// TIA Portal project "Practica3Equipo" (V16)

(* hardware
DEVICE "S7300/ET200M station_1"  S7-300 station
   slot 0: "Rail_0"  Rail  6ES7 390-1***0-0AA0
   slot 2: "PLC_1"  CPU 314  6ES7 314-1AG13-0AB0  V2.6
      slot 0: "MPI interface_1"  X1
*)

// ===== PLC "PLC_1"  CPU 314 =====

VAR_GLOBAL   // PLC tag table "Estados"
   "E0" AT %M0.0 : Bool;
   "E1" AT %M0.1 : Bool;
   "E2" AT %M0.2 : Bool;
   "E3" AT %M0.3 : Bool;
   "E4" AT %M0.4 : Bool;
   "E5" AT %M0.5 : Bool;
   "E6" AT %M0.6 : Bool;
   "E7" AT %M0.7 : Bool;
   "E8" AT %M1.0 : Bool;
   "E9" AT %M1.1 : Bool;
   "E10" AT %M1.2 : Bool;
   "E11" AT %M1.3 : Bool;
   "E12" AT %M1.4 : Bool;
   "E13" AT %M1.5 : Bool;
   "E14" AT %M1.6 : Bool;
   "E15" AT %M1.7 : Bool;
   "E16" AT %M2.0 : Bool;
   "E17" AT %M2.1 : Bool;
   "E18" AT %M2.2 : Bool;
   "E19" AT %M2.3 : Bool;
END_VAR

VAR_GLOBAL   // PLC tag table "Inputs"
   "P3inWork" AT %I10.0 : Bool;
   "P3inHome" AT %I10.1 : Bool;
   "P3engaged" AT %I10.2 : Bool;
   "RStation1" AT %I10.3 : Bool;
   "RStation2" AT %I10.4 : Bool;
   "Lightbarrier" AT %I10.5 : Bool;
   "inPlace3" AT %I10.6 : Bool;
   "inPlace4" AT %I10.7 : Bool;
   "P1inWork" AT %I11.0 : Bool;
   "P1inHome" AT %I11.1 : Bool;
   "P2inWork" AT %I11.2 : Bool;
   "P2inHome" AT %I11.3 : Bool;
   "P1engaged" AT %I11.4 : Bool;
   "P2engaged" AT %I11.5 : Bool;
   "inPlace1" AT %I11.6 : Bool;
   "inPlace2" AT %I11.7 : Bool;
   "chainMagnet" AT %I13.6 : Bool;
END_VAR

VAR_GLOBAL   // PLC tag table "Outputs"
   "Chain" AT %Q11.0 : Bool;
   "Belt" AT %Q11.1 : Bool;
   "P1toWork" AT %Q11.2 : Bool;
   "P1toHome" AT %Q11.3 : Bool;
   "P2toWork" AT %Q11.4 : Bool;
   "P2toHome" AT %Q11.5 : Bool;
   "P3toWork" AT %Q11.6 : Bool;
   "P3toHome" AT %Q11.7 : Bool;
END_VAR

FUNCTION "Secuencial" : Void   // FC1, LAD
{ S7_Optimized_Access := 'FALSE' }
VERSION : 0.1
   VAR_TEMP   // added for the SCL form of the ladder/FBD networks
      _w1 : Bool;
   END_VAR
BEGIN

REGION Network 1
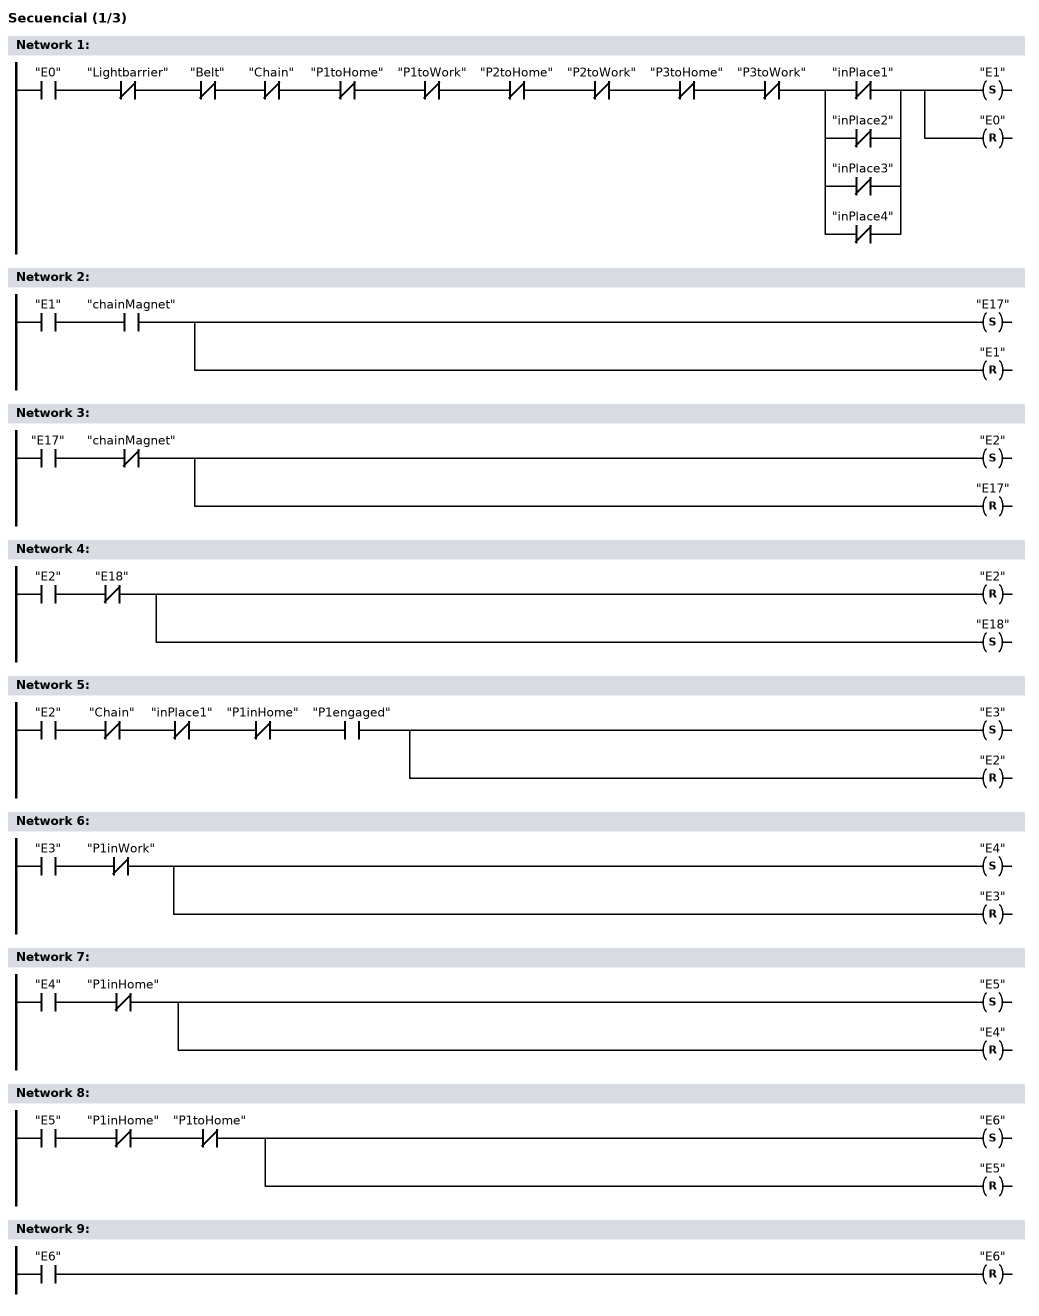
   RUNG wire#powerrail
      Contact( "E0" )
      I_Contact( "Lightbarrier" )
      I_Contact( "Belt" )
      I_Contact( "Chain" )
      I_Contact( "P1toHome" )
      I_Contact( "P1toWork" )
      I_Contact( "P2toHome" )
      I_Contact( "P2toWork" )
      I_Contact( "P3toHome" )
      I_Contact( "P3toWork" )
      wire#w1
      I_Contact( "inPlace1" )
      wire#w2
      S_Coil( "E1" )
   END_RUNG
   RUNG wire#w1
      I_Contact( "inPlace2" )
   END_RUNG wire#w2
   RUNG wire#w1
      I_Contact( "inPlace3" )
   END_RUNG wire#w2
   RUNG wire#w1
      I_Contact( "inPlace4" )
   END_RUNG wire#w2
   RUNG wire#w2
      R_Coil( "E0" )
   END_RUNG
   // the same network as SCL:
   IF "E0" AND NOT "Lightbarrier" AND NOT "Belt" AND NOT "Chain" AND NOT "P1toHome" AND NOT "P1toWork" AND NOT "P2toHome" AND NOT "P2toWork" AND NOT "P3toHome" AND NOT "P3toWork" AND (NOT "inPlace1" OR NOT "inPlace2" OR NOT "inPlace3" OR NOT "inPlace4") THEN
       "E1" := TRUE;
       "E0" := FALSE;
   END_IF;
END_REGION

REGION Network 2
   RUNG wire#powerrail
      Contact( "E1" )
      Contact( "chainMagnet" )
      wire#w1
      S_Coil( "E17" )
   END_RUNG
   RUNG wire#w1
      R_Coil( "E1" )
   END_RUNG
   // the same network as SCL:
   IF "E1" AND "chainMagnet" THEN
       "E17" := TRUE;
       "E1" := FALSE;
   END_IF;
END_REGION

REGION Network 3
   RUNG wire#powerrail
      Contact( "E17" )
      I_Contact( "chainMagnet" )
      wire#w1
      S_Coil( "E2" )
   END_RUNG
   RUNG wire#w1
      R_Coil( "E17" )
   END_RUNG
   // the same network as SCL:
   IF "E17" AND NOT "chainMagnet" THEN
       "E2" := TRUE;
       "E17" := FALSE;
   END_IF;
END_REGION

REGION Network 4
   RUNG wire#powerrail
      Contact( "E2" )
      I_Contact( "E18" )
      wire#w1
      R_Coil( "E2" )
   END_RUNG
   RUNG wire#w1
      S_Coil( "E18" )
   END_RUNG
   // the same network as SCL:
   #_w1 := "E2" AND NOT "E18";
   IF #_w1 THEN
       "E2" := FALSE;
       "E18" := TRUE;
   END_IF;
END_REGION

REGION Network 5
   RUNG wire#powerrail
      Contact( "E2" )
      I_Contact( "Chain" )
      I_Contact( "inPlace1" )
      I_Contact( "P1inHome" )
      Contact( "P1engaged" )
      wire#w1
      S_Coil( "E3" )
   END_RUNG
   RUNG wire#w1
      R_Coil( "E2" )
   END_RUNG
   // the same network as SCL:
   IF "E2" AND NOT "Chain" AND NOT "inPlace1" AND NOT "P1inHome" AND "P1engaged" THEN
       "E3" := TRUE;
       "E2" := FALSE;
   END_IF;
END_REGION

REGION Network 6
   RUNG wire#powerrail
      Contact( "E3" )
      I_Contact( "P1inWork" )
      wire#w1
      S_Coil( "E4" )
   END_RUNG
   RUNG wire#w1
      R_Coil( "E3" )
   END_RUNG
   // the same network as SCL:
   IF "E3" AND NOT "P1inWork" THEN
       "E4" := TRUE;
       "E3" := FALSE;
   END_IF;
END_REGION

REGION Network 7
   RUNG wire#powerrail
      Contact( "E4" )
      I_Contact( "P1inHome" )
      wire#w1
      S_Coil( "E5" )
   END_RUNG
   RUNG wire#w1
      R_Coil( "E4" )
   END_RUNG
   // the same network as SCL:
   IF "E4" AND NOT "P1inHome" THEN
       "E5" := TRUE;
       "E4" := FALSE;
   END_IF;
END_REGION

REGION Network 8
   RUNG wire#powerrail
      Contact( "E5" )
      I_Contact( "P1inHome" )
      I_Contact( "P1toHome" )
      wire#w1
      S_Coil( "E6" )
   END_RUNG
   RUNG wire#w1
      R_Coil( "E5" )
   END_RUNG
   // the same network as SCL:
   IF "E5" AND NOT "P1inHome" AND NOT "P1toHome" THEN
       "E6" := TRUE;
       "E5" := FALSE;
   END_IF;
END_REGION

REGION Network 9
   RUNG wire#powerrail
      Contact( "E6" )
      R_Coil( "E6" )
   END_RUNG
   // the same network as SCL:
   IF "E6" THEN "E6" := FALSE; END_IF;
END_REGION

REGION Network 10
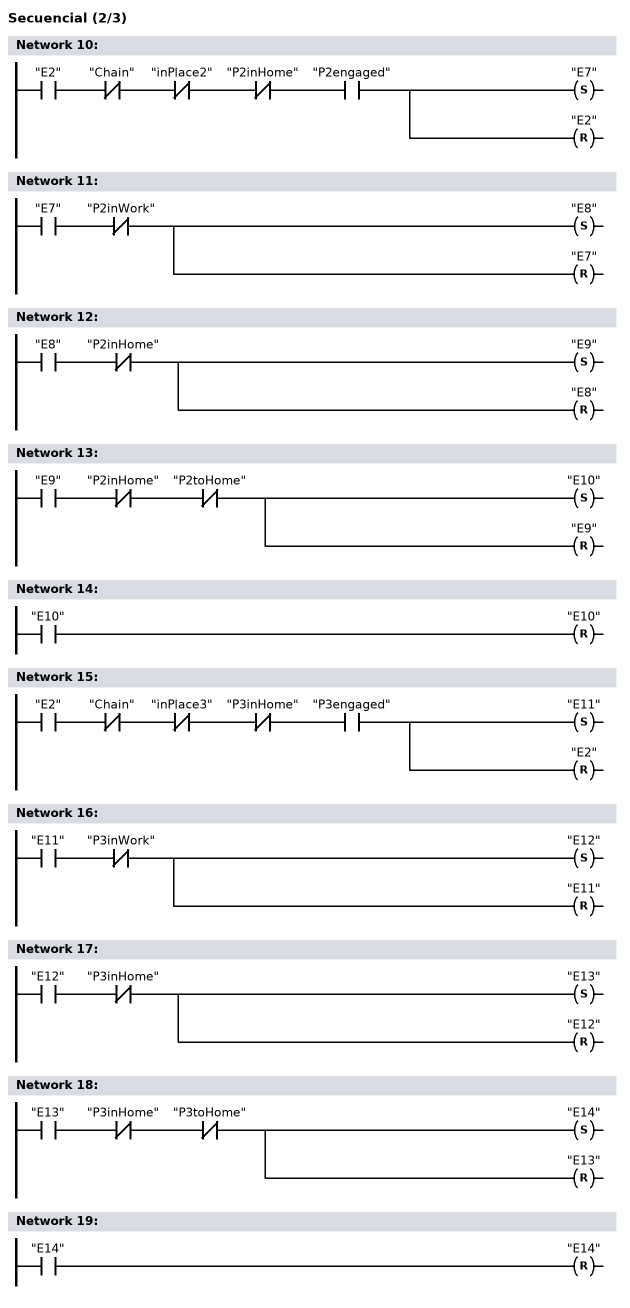
   RUNG wire#powerrail
      Contact( "E2" )
      I_Contact( "Chain" )
      I_Contact( "inPlace2" )
      I_Contact( "P2inHome" )
      Contact( "P2engaged" )
      wire#w1
      S_Coil( "E7" )
   END_RUNG
   RUNG wire#w1
      R_Coil( "E2" )
   END_RUNG
   // the same network as SCL:
   IF "E2" AND NOT "Chain" AND NOT "inPlace2" AND NOT "P2inHome" AND "P2engaged" THEN
       "E7" := TRUE;
       "E2" := FALSE;
   END_IF;
END_REGION

REGION Network 11
   RUNG wire#powerrail
      Contact( "E7" )
      I_Contact( "P2inWork" )
      wire#w1
      S_Coil( "E8" )
   END_RUNG
   RUNG wire#w1
      R_Coil( "E7" )
   END_RUNG
   // the same network as SCL:
   IF "E7" AND NOT "P2inWork" THEN
       "E8" := TRUE;
       "E7" := FALSE;
   END_IF;
END_REGION

REGION Network 12
   RUNG wire#powerrail
      Contact( "E8" )
      I_Contact( "P2inHome" )
      wire#w1
      S_Coil( "E9" )
   END_RUNG
   RUNG wire#w1
      R_Coil( "E8" )
   END_RUNG
   // the same network as SCL:
   IF "E8" AND NOT "P2inHome" THEN
       "E9" := TRUE;
       "E8" := FALSE;
   END_IF;
END_REGION

REGION Network 13
   RUNG wire#powerrail
      Contact( "E9" )
      I_Contact( "P2inHome" )
      I_Contact( "P2toHome" )
      wire#w1
      S_Coil( "E10" )
   END_RUNG
   RUNG wire#w1
      R_Coil( "E9" )
   END_RUNG
   // the same network as SCL:
   IF "E9" AND NOT "P2inHome" AND NOT "P2toHome" THEN
       "E10" := TRUE;
       "E9" := FALSE;
   END_IF;
END_REGION

REGION Network 14
   RUNG wire#powerrail
      Contact( "E10" )
      R_Coil( "E10" )
   END_RUNG
   // the same network as SCL:
   IF "E10" THEN "E10" := FALSE; END_IF;
END_REGION

REGION Network 15
   RUNG wire#powerrail
      Contact( "E2" )
      I_Contact( "Chain" )
      I_Contact( "inPlace3" )
      I_Contact( "P3inHome" )
      Contact( "P3engaged" )
      wire#w1
      S_Coil( "E11" )
   END_RUNG
   RUNG wire#w1
      R_Coil( "E2" )
   END_RUNG
   // the same network as SCL:
   IF "E2" AND NOT "Chain" AND NOT "inPlace3" AND NOT "P3inHome" AND "P3engaged" THEN
       "E11" := TRUE;
       "E2" := FALSE;
   END_IF;
END_REGION

REGION Network 16
   RUNG wire#powerrail
      Contact( "E11" )
      I_Contact( "P3inWork" )
      wire#w1
      S_Coil( "E12" )
   END_RUNG
   RUNG wire#w1
      R_Coil( "E11" )
   END_RUNG
   // the same network as SCL:
   IF "E11" AND NOT "P3inWork" THEN
       "E12" := TRUE;
       "E11" := FALSE;
   END_IF;
END_REGION

REGION Network 17
   RUNG wire#powerrail
      Contact( "E12" )
      I_Contact( "P3inHome" )
      wire#w1
      S_Coil( "E13" )
   END_RUNG
   RUNG wire#w1
      R_Coil( "E12" )
   END_RUNG
   // the same network as SCL:
   IF "E12" AND NOT "P3inHome" THEN
       "E13" := TRUE;
       "E12" := FALSE;
   END_IF;
END_REGION

REGION Network 18
   RUNG wire#powerrail
      Contact( "E13" )
      I_Contact( "P3inHome" )
      I_Contact( "P3toHome" )
      wire#w1
      S_Coil( "E14" )
   END_RUNG
   RUNG wire#w1
      R_Coil( "E13" )
   END_RUNG
   // the same network as SCL:
   IF "E13" AND NOT "P3inHome" AND NOT "P3toHome" THEN
       "E14" := TRUE;
       "E13" := FALSE;
   END_IF;
END_REGION

REGION Network 19
   RUNG wire#powerrail
      Contact( "E14" )
      R_Coil( "E14" )
   END_RUNG
   // the same network as SCL:
   IF "E14" THEN "E14" := FALSE; END_IF;
END_REGION

REGION Network 20
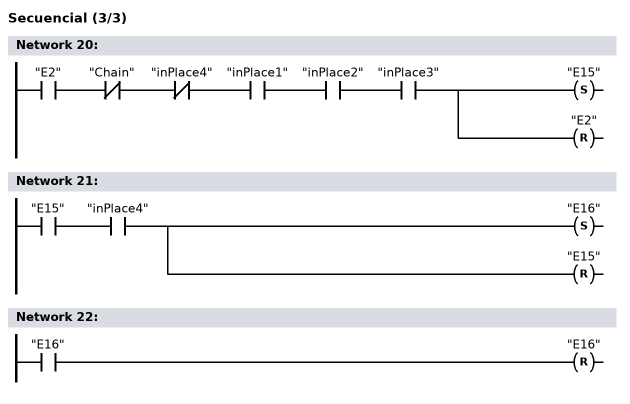
   RUNG wire#powerrail
      Contact( "E2" )
      I_Contact( "Chain" )
      I_Contact( "inPlace4" )
      Contact( "inPlace1" )
      Contact( "inPlace2" )
      Contact( "inPlace3" )
      wire#w1
      S_Coil( "E15" )
   END_RUNG
   RUNG wire#w1
      R_Coil( "E2" )
   END_RUNG
   // the same network as SCL:
   IF "E2" AND NOT "Chain" AND NOT "inPlace4" AND "inPlace1" AND "inPlace2" AND "inPlace3" THEN
       "E15" := TRUE;
       "E2" := FALSE;
   END_IF;
END_REGION

REGION Network 21
   RUNG wire#powerrail
      Contact( "E15" )
      Contact( "inPlace4" )
      wire#w1
      S_Coil( "E16" )
   END_RUNG
   RUNG wire#w1
      R_Coil( "E15" )
   END_RUNG
   // the same network as SCL:
   IF "E15" AND "inPlace4" THEN
       "E16" := TRUE;
       "E15" := FALSE;
   END_IF;
END_REGION

REGION Network 22
   RUNG wire#powerrail
      Contact( "E16" )
      R_Coil( "E16" )
   END_RUNG
   // the same network as SCL:
   IF "E16" THEN "E16" := FALSE; END_IF;
END_REGION
END_FUNCTION

FUNCTION "Combinacional" : Void   // FC2, LAD
{ S7_Optimized_Access := 'FALSE' }
VERSION : 0.1
BEGIN

REGION Network 1
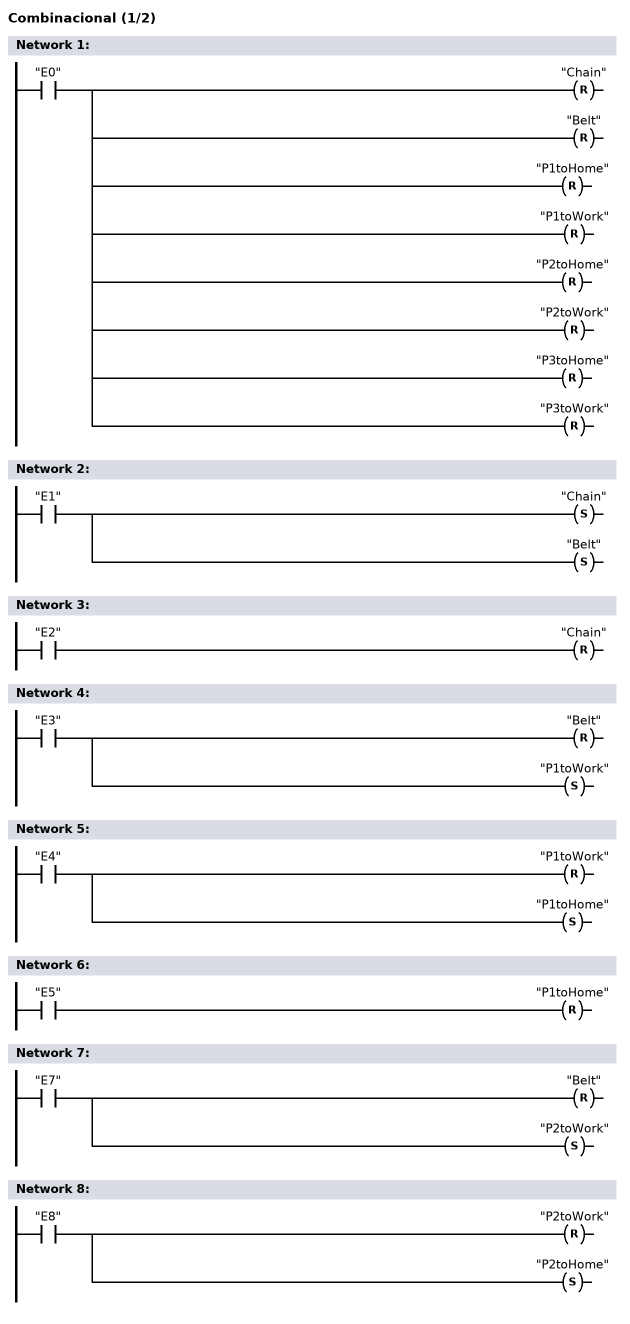
   RUNG wire#powerrail
      Contact( "E0" )
      wire#w1
      R_Coil( "Chain" )
   END_RUNG
   RUNG wire#w1
      R_Coil( "Belt" )
   END_RUNG
   RUNG wire#w1
      R_Coil( "P1toHome" )
   END_RUNG
   RUNG wire#w1
      R_Coil( "P1toWork" )
   END_RUNG
   RUNG wire#w1
      R_Coil( "P2toHome" )
   END_RUNG
   RUNG wire#w1
      R_Coil( "P2toWork" )
   END_RUNG
   RUNG wire#w1
      R_Coil( "P3toHome" )
   END_RUNG
   RUNG wire#w1
      R_Coil( "P3toWork" )
   END_RUNG
   // the same network as SCL:
   IF "E0" THEN
       "Chain" := FALSE;
       "Belt" := FALSE;
       "P1toHome" := FALSE;
       "P1toWork" := FALSE;
       "P2toHome" := FALSE;
       "P2toWork" := FALSE;
       "P3toHome" := FALSE;
       "P3toWork" := FALSE;
   END_IF;
END_REGION

REGION Network 2
   RUNG wire#powerrail
      Contact( "E1" )
      wire#w1
      S_Coil( "Chain" )
   END_RUNG
   RUNG wire#w1
      S_Coil( "Belt" )
   END_RUNG
   // the same network as SCL:
   IF "E1" THEN
       "Chain" := TRUE;
       "Belt" := TRUE;
   END_IF;
END_REGION

REGION Network 3
   RUNG wire#powerrail
      Contact( "E2" )
      R_Coil( "Chain" )
   END_RUNG
   // the same network as SCL:
   IF "E2" THEN "Chain" := FALSE; END_IF;
END_REGION

REGION Network 4
   RUNG wire#powerrail
      Contact( "E3" )
      wire#w1
      R_Coil( "Belt" )
   END_RUNG
   RUNG wire#w1
      S_Coil( "P1toWork" )
   END_RUNG
   // the same network as SCL:
   IF "E3" THEN
       "Belt" := FALSE;
       "P1toWork" := TRUE;
   END_IF;
END_REGION

REGION Network 5
   RUNG wire#powerrail
      Contact( "E4" )
      wire#w1
      R_Coil( "P1toWork" )
   END_RUNG
   RUNG wire#w1
      S_Coil( "P1toHome" )
   END_RUNG
   // the same network as SCL:
   IF "E4" THEN
       "P1toWork" := FALSE;
       "P1toHome" := TRUE;
   END_IF;
END_REGION

REGION Network 6
   RUNG wire#powerrail
      Contact( "E5" )
      R_Coil( "P1toHome" )
   END_RUNG
   // the same network as SCL:
   IF "E5" THEN "P1toHome" := FALSE; END_IF;
END_REGION

REGION Network 7
   RUNG wire#powerrail
      Contact( "E7" )
      wire#w1
      R_Coil( "Belt" )
   END_RUNG
   RUNG wire#w1
      S_Coil( "P2toWork" )
   END_RUNG
   // the same network as SCL:
   IF "E7" THEN
       "Belt" := FALSE;
       "P2toWork" := TRUE;
   END_IF;
END_REGION

REGION Network 8
   RUNG wire#powerrail
      Contact( "E8" )
      wire#w1
      R_Coil( "P2toWork" )
   END_RUNG
   RUNG wire#w1
      S_Coil( "P2toHome" )
   END_RUNG
   // the same network as SCL:
   IF "E8" THEN
       "P2toWork" := FALSE;
       "P2toHome" := TRUE;
   END_IF;
END_REGION

REGION Network 9
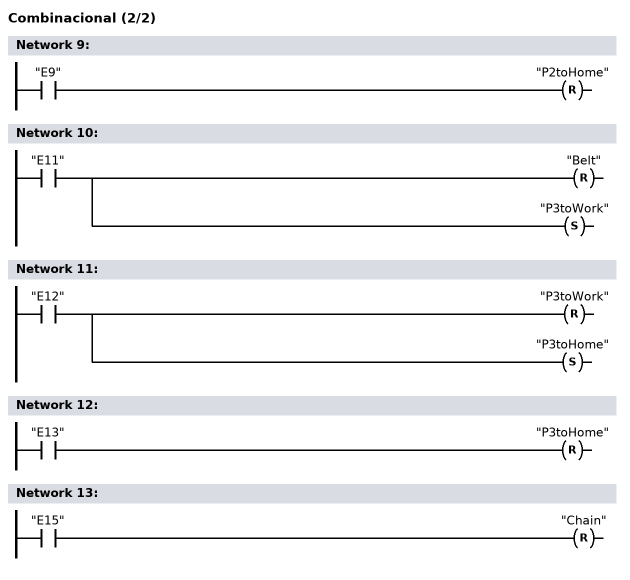
   RUNG wire#powerrail
      Contact( "E9" )
      R_Coil( "P2toHome" )
   END_RUNG
   // the same network as SCL:
   IF "E9" THEN "P2toHome" := FALSE; END_IF;
END_REGION

REGION Network 10
   RUNG wire#powerrail
      Contact( "E11" )
      wire#w1
      R_Coil( "Belt" )
   END_RUNG
   RUNG wire#w1
      S_Coil( "P3toWork" )
   END_RUNG
   // the same network as SCL:
   IF "E11" THEN
       "Belt" := FALSE;
       "P3toWork" := TRUE;
   END_IF;
END_REGION

REGION Network 11
   RUNG wire#powerrail
      Contact( "E12" )
      wire#w1
      R_Coil( "P3toWork" )
   END_RUNG
   RUNG wire#w1
      S_Coil( "P3toHome" )
   END_RUNG
   // the same network as SCL:
   IF "E12" THEN
       "P3toWork" := FALSE;
       "P3toHome" := TRUE;
   END_IF;
END_REGION

REGION Network 12
   RUNG wire#powerrail
      Contact( "E13" )
      R_Coil( "P3toHome" )
   END_RUNG
   // the same network as SCL:
   IF "E13" THEN "P3toHome" := FALSE; END_IF;
END_REGION

REGION Network 13
   RUNG wire#powerrail
      Contact( "E15" )
      R_Coil( "Chain" )
   END_RUNG
   // the same network as SCL:
   IF "E15" THEN "Chain" := FALSE; END_IF;
END_REGION
END_FUNCTION

ORGANIZATION_BLOCK "Main"   // OB1, LAD
TITLE = "Main Program Sweep (Cycle)"
{ S7_Optimized_Access := 'FALSE' }
VERSION : 0.1
   VAR_TEMP
      OB1_EV_CLASS : Byte;   // Bits 0-3 = 1 (Coming event), Bits 4-7 = 1 (Event class 1)
      OB1_SCAN_1 : Byte;   // 1 (Cold restart scan 1 of OB 1), 3 (Scan 2-n of OB 1)
      OB1_PRIORITY : Byte;   // Priority of OB Execution
      OB1_OB_NUMBR : Byte;   // 1 (Organization block 1, OB1)
      OB1_RESERVED_1 : Byte;   // Reserved for system
      OB1_RESERVED_2 : Byte;   // Reserved for system
      OB1_PREV_CYCLE : Int;   // Cycle time of previous OB1 scan (milliseconds)
      OB1_MIN_CYCLE : Int;   // Minimum cycle time of OB1 (milliseconds)
      OB1_MAX_CYCLE : Int;   // Maximum cycle time of OB1 (milliseconds)
      OB1_DATE_TIME : Date_And_Time;   // Date and time OB1 started
   END_VAR
BEGIN

REGION Network 1
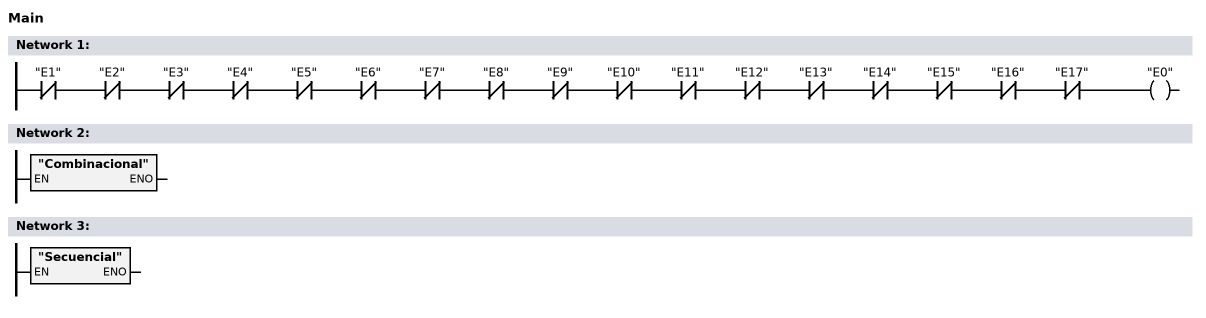
   RUNG wire#powerrail
      I_Contact( "E1" )
      I_Contact( "E2" )
      I_Contact( "E3" )
      I_Contact( "E4" )
      I_Contact( "E5" )
      I_Contact( "E6" )
      I_Contact( "E7" )
      I_Contact( "E8" )
      I_Contact( "E9" )
      I_Contact( "E10" )
      I_Contact( "E11" )
      I_Contact( "E12" )
      I_Contact( "E13" )
      I_Contact( "E14" )
      I_Contact( "E15" )
      I_Contact( "E16" )
      I_Contact( "E17" )
      Coil( "E0" )
   END_RUNG
   // the same network as SCL:
   "E0" := NOT "E1" AND NOT "E2" AND NOT "E3" AND NOT "E4" AND NOT "E5" AND NOT "E6" AND NOT "E7" AND NOT "E8" AND NOT "E9" AND NOT "E10" AND NOT "E11" AND NOT "E12" AND NOT "E13" AND NOT "E14" AND NOT "E15" AND NOT "E16" AND NOT "E17";
END_REGION

REGION Network 2
   RUNG wire#powerrail
      "Combinacional"()
   END_RUNG
   // the same network as SCL:
   "Combinacional"();
END_REGION

REGION Network 3
   RUNG wire#powerrail
      "Secuencial"()
   END_RUNG
   // the same network as SCL:
   "Secuencial"();
END_REGION
END_ORGANIZATION_BLOCK